TYPE ST_LivingRoomDevices :
STRUCT

	sShellyLight						: ST_StatusShellyOnePM;	
	
END_STRUCT
END_TYPE

(* stored: Version 1.1.0.1, ProductVersion 3.1.4024.12
   DUT ST_LivingRoomDevices: Id {cd3954fc-b543-4deb-808a-780d2dd2d086} *)
